{attribute 'qualified_only'}
{attribute 'to_string'}
TYPE ZAppStep :
(
  Undefined := 0
  
  ,BootBegin
  ,BootLoadDefaultData
  ,BootEnd
  ,BootFaultBegin
  ,BootFaultEnd 
  ,RunningBegin
  ,RunningEnd   
);
END_TYPE

(* stored: Version 1.1.0.1
   DUT ZAppStep: Id {3ff07284-b4bd-4d3b-9b75-6656cd4dc9aa} *)
